TYPE DUT_StatePMPSEpicsInterface EXTENDS DUT_StateEpicsInterface :
(*
    This data structure contains the standard EPICS connection points for the state movers.

    See DUT_StateEpicsInterface, this is an extension to add the PMPS settings.
*)
STRUCT
    // TRUE if the arbiter is enabled, FALSE if it is disabled.
    {attribute 'pytmc' := '
        pv: PMPS:ARB:ENABLE
        io: io
    '}
    bArbiterEnabled: BOOL;
    // TRUE if we're in maintenance mode (Fast fault, free motion), FALSE otherwise.
    {attribute 'pytmc' := '
        pv: PMPS:MAINT
        io: io
    '}
    bMaintMode: BOOL;
    // The database entry for the transition state. This should always be present.
    {attribute 'pytmc' := '
        pv: PMPS:TRANS
        io: i
    '}
    stTransitionDb: ST_DbStateParams;
END_STRUCT
END_TYPE

(* stored: Version 1.1.0.1, ProductVersion 3.1.4022.18
   DUT DUT_StatePMPSEpicsInterface: Id {fe26de4c-1758-435b-90a9-da23c711b889} *)
